{attribute 'qualified_only'}
{attribute 'strict'}
TYPE E_MotorVFD :
(
	enum_member := 0
);
END_TYPE

(* stored: Version 1.1.0.1, ProductVersion 3.1.4024.12
   DUT E_MotorVFD: Id {0551637e-c366-4f52-a19a-1be9f2201408} *)
